(* Logix 5000 project; controller Uidaho_Factory vendor 1 type 14 code 165 rev 38.11; software revision 38.00 *)

TASK Heartbeat (periodic, rate 10000 ms, priority 10, watchdog 500 ms) : Heartbeat
TASK MainTask (continuous, watchdog 500 ms) : MainProgram

MODULES
   Local : vendor 1 type 14 code 165 (ICP 0, rev 38.11)
      Slot_3_Input : vendor 1 type 7 code 6 (ICP 3, rev 2.2, Input RPI 20 ms)
           Local:3:I.Data.3   // MPO - I8 = Reference switch vacuum (position oven)
           Local:3:I.Data.0   // MPO - I5 = Reference switch vacuum (position turn-table)
           Local:3:I.Data.5   // VGR - I1 = Reference switch vertical axis
           Local:3:I.Data.1   // MPO - I6 = Reference switch oven feeder inside
           Local:3:I.Data.2   // MPO - I7 = Reference switch oven feeder outside
           Local:3:I.Data.10   // SLD - I3 = Light barrier behind color sensor
           Local:3:I.Data.4   // MPO - I9 = Light barrier oven
           Local:3:I.Data.12   // SLD - I6 = Light barrier red
           Local:3:I.Data.13   // SLD - I7 = Light barrier blue
           Local:3:I.Data.8   // SLD - I1 = Pulse counter
           Local:3:I.Data.11   // SLD - I5 = Light barrier white
           Local:3:I.Data.9   // SLD - I2 = Light barrier inlet
           Local:3:I.Data.14   // SSC - I1 = Reference switch vertical axis
           Local:3:I.Data.6   // VGR - I2 = Reference switch horizontal axis
           Local:3:I.Data.7   // VGR - I3 = Reference switch rotate
           Local:3:I.Data.15   // SSC - I2 = Reference switch horizontal axis
      Slot_4_Input : vendor 1 type 7 code 6 (ICP 4, rev 2.2, Input RPI 20 ms)
           Local:4:I.Data.2   // SSC - B1 = Encoder vertical axis impulse 1
           Local:4:I.Data.1   // SSC - I4 = Light barrier behind color sensor
           Local:4:I.Data.4   // SSC - B3 = Encoder horizontal axis impulse 1
           Local:4:I.Data.5   // SSC - B4 = Encoder horizontal axis impulse 2
           Local:4:I.Data.3   // SSC - B2 = Encoder vertical axis impulse 2
           Local:4:I.Data.0   // SSC - I3 = Light barrier inlet
      Slot_2_Input : vendor 1 type 7 code 6 (ICP 2, rev 2.2, Input RPI 20 ms)
           Local:2:I.Data.15   // MPO - I4 = Reference switch turn-table (position saw)
           Local:2:I.Data.12   // MPO - I1 = Reference switch turn-table (position vacuum)
           Local:2:I.Data.3   // HBW - I4 = Reference switch vertical axis
           Local:2:I.Data.13   // MPO - I2 = Reference switch turn-table (position belt)
           Local:2:I.Data.14   // MPO - I3 = Light barrier end of conveyor belt
           Local:2:I.Data.10   // HBW - I5 = Reference switch cantilever front
           Local:2:I.Data.8   // HBW - B1 = Encoder horizontal axis impulse 1
           Local:2:I.Data.4   // HBW - A1 = Trail sensor (signal 1, lower)
           Local:2:I.Data.5   // HBW - A2 = Trail sensor (signal 2, upper)
           Local:2:I.Data.9   // HBW - B2 = Encoder horizontal axis impulse 2
           Local:2:I.Data.6   // HBW - B3 = Encoder vertical axis impulse 1
           Local:2:I.Data.7   // HBW - B4 = Encoder vertical axis impulse 2
           Local:2:I.Data.0   // HBW - I1 = Reference switch horizontal axis
           Local:2:I.Data.11   // HBW - I6 = Reference switch cantilever back
           Local:2:I.Data.2   // HBW - I3 = Light barrier outside
           Local:2:I.Data.1   // HBW - I2 = Light barrier inside
      Slot_1_Input : vendor 1 type 7 code 386 (ICP 1, rev 1.11, Output RPI 20 ms)
           Local:1:I.Pt[2].Data   // VGR - B3 = Encoder horizontal axis impulse 1
           Local:1:I.Pt[4].Data   // VGR - B5 = Encoder rotate impulse 1
           Local:1:I.Pt[5].Data   // VGR - B6 = Encoder rotate impulse 2
           Local:1:I.Pt[0].Data   // VGR - B1 = Encoder vertical axis impulse 1
           Local:1:I.Pt[3].Data   // VGR - B4 = Encoder horizontal axis impulse 2
           Local:1:I.Pt[1].Data   // VGR - B2 = Encoder vertical axis impulse 2
      Slot_6_Output : 1756-OB32 (ICP 6, rev 2.4, Output RPI 20 ms)
           Local:6:O.Data.17   // SSC - Q3 = Motor M2 horizontal axis backward
           Local:6:O.Data.20   // MPO - Q5 = Motor M4 oven feeder retract
           Local:6:O.Data.28   // VGR - Q3 = Motor M2 horizontal axis retract
           Local:6:O.Data.22   // MPO - Q2 = Motor M1 turn-table counterclockwise
           Local:6:O.Data.25   // MPO - Q10 = Compressor
           Local:6:O.Data.18   // SSC - Q4 = Motor M2 horizontal axis forward
           Local:6:O.Data.29   // VGR - Q4 = Motor M2 horizontal axis extend
           Local:6:O.Data.1   // HBW - Q6 = Motor M3 vertical axis upward
           Local:6:O.Data.10   // VGR - Q1 = Motor M1 vertical axis up
           Local:6:O.Data.11   // VGR - Q2 = Motor M1 vertical axis down
           Local:6:O.Data.9   // MPO - Q14 = Valve feeder
           Local:6:O.Data.16   // SSC - Q2 = Motor M1 vertical axis down
           Local:6:O.Data.2   // HBW - Q7 = Motor M4 cantilever forward
           Local:6:O.Data.30   // VGR - Q5 = Motor M3 rotate clockwise
           Local:6:O.Data.0   // HBW - Q5 = Motor M3 vertical axis downward
           Local:6:O.Data.4   // SSC = PWM Motor M1 vertical axis
           Local:6:O.Data.31   // VGR - Q6 = Motor M3 rotate counterclockwise
           Local:6:O.Data.3   // HBW - Q8 = Motor M4 cantilever backward
           Local:6:O.Data.14   // SLD - Q1 = Motor M1conveyor belt
           Local:6:O.Data.7   // MPO - Q8 = Motor M5 vacuum towards turn-table
           Local:6:O.Data.23   // MPO - Q3 = Motor M2 conveyor belt forward
           Local:6:O.Data.5   // SSC = PWM Motor M2 horizontal axis
           Local:6:O.Data.21   // MPO - Q1 = Motor M1 turn-table clockwise
           Local:6:O.Data.26   // MPO - Q11 = Valve vacuum
           Local:6:O.Data.19   // SSC - Q5 = LED Green
           Local:6:O.Data.27   // MPO - Q12 = Valve lowering
           Local:6:O.Data.13   // VGR - Q8 = Valve vacuum
           Local:6:O.Data.12   // VGR - Q7 = Compressor
           Local:6:O.Data.15   // SLD - Q2 = Compressor
           Local:6:O.Data.24   // MPO - Q9 = Light oven
           Local:6:O.Data.6   // QW_MPO_PWM_TurnTable_M1
           Local:6:O.Data.8   // MPO - Q13 = Valve oven door
      Slot_7_Output : 1756-OB32 (ICP 7, rev 3.2, Output RPI 20 ms)
           Local:7:O.Data.19   // VGR = PWM Motor M2 horizontal axis
           Local:7:O.Data.0   // SLD - Q3 = Valve first ejector (white)
           Local:7:O.Data.18   // VGR = PWM Motor M1 vertical axis
           Local:7:O.Data.3   // SSC - Q1 = Motor M1 vertical axis up
           Local:7:O.Data.1   // SLD - Q4 = Valve second ejector (red)
           Local:7:O.Data.15   // HBW = PWM Motor M2 horizontal axis
           Local:7:O.Data.12   // HBW - Q3 = Motor M2 horizontal towards rack
           Local:7:O.Data.13   // HBW - Q4 = Motor M2 horizontal towards conveyor belt
           Local:7:O.Data.8   // MPO - Q6 = Motor M4 oven feeder extend
           Local:7:O.Data.10   // HBW - Q1 = Motor M1 conveyor belt forward
           Local:7:O.Data.11   // HBW - Q2 = Motor M1 conveyor belt backward
           Local:7:O.Data.17   // HBW = PWM Motor M4 cantilever
           Local:7:O.Data.2   // SLD - Q5 = Valve third ejector (blue)
           Local:7:O.Data.21   // MPO = PWM Motor M5 vacuum
           Local:7:O.Data.9   // MPO - Q7 = Motor M5 vacuum towards oven
           Local:7:O.Data.20   // VGR = PWM Motor M3 rotate axis
           Local:7:O.Data.14   // HBW = PWM Motor M1 conveyor belt
           Local:7:O.Data.16   // HBW = PWM Motor M3 vertical axis
           Local:7:O.Data.6   // SSC - Q8 = LED Red Online
           Local:7:O.Data.7   // MPO - Q4 = Motor M3 saw
           Local:7:O.Data.4   // SSC - Q6 = LED Yellow
           Local:7:O.Data.5   // Turn on Motor Rotation Clockwise
      Slot_5_Input : 1756-IF8 (ICP 5, rev 1.5, Input RPI 100 ms)
           Local:5:I.Ch1Data   // SLD - A1 = Color sensor
           Local:5:I.Ch0Data   // SSC - A4 = Color sensor
END_MODULES

ADD_ON_INSTRUCTION PWM_Out   (* revision 1.0, ExecutePrescan *)
VAR_OUTPUT
   PWM_Pin : BOOL; {required}
END_VAR
VAR_INPUT
   Duty_Cycle : DINT; {required}
   Frequency_Hz : DINT; {required}
END_VAR
VAR
   PWM_Timer_On : TIMER; {access None}
   PWM_Timer_Off : TIMER; {access None}
   Duty_Cycle_Scaler : REAL; {access None}
   Frequency_Ms : REAL := 60.0; {access None}
   Fault_Bit : BOOL; {access None}
END_VAR

ROUTINE Logic   (* ladder *)
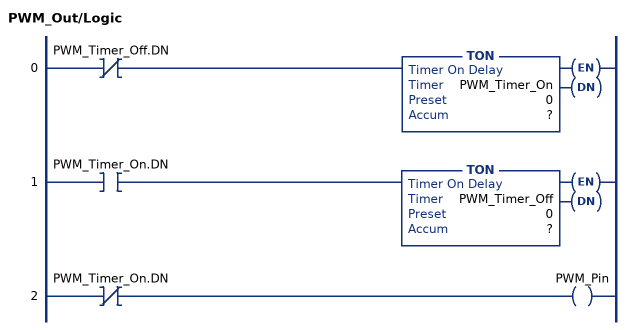
   0: XIO(PWM_Timer_Off.DN)TON(PWM_Timer_On,?,?);
   1: XIC(PWM_Timer_On.DN)TON(PWM_Timer_Off,?,?);
   2: XIO(PWM_Timer_On.DN)OTE(PWM_Pin);
END_ROUTINE

ROUTINE Prescan   (* ladder *)
// Perform Calculations for PWM Timing
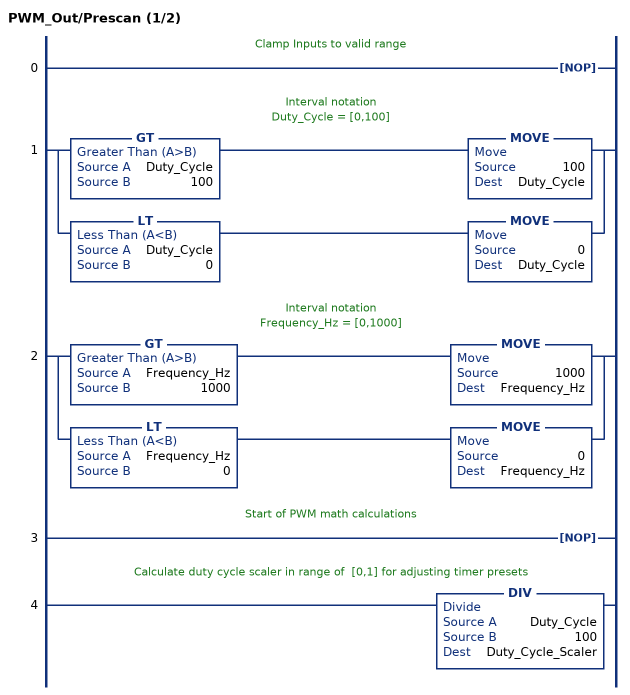
   // Clamp Inputs to valid range
   0: NOP();
   // Interval notation
   // Duty_Cycle = [0,100]
   1: [GT(Duty_Cycle,100) MOVE(100,Duty_Cycle) ,LT(Duty_Cycle,0) MOVE(0,Duty_Cycle) ];
   // Interval notation
   // Frequency_Hz = [0,1000]
   2: [GT(Frequency_Hz,1000) MOVE(1000,Frequency_Hz) ,LT(Frequency_Hz,0) MOVE(0,Frequency_Hz) ];
   // Start of PWM math calculations
   3: NOP();
   // Calculate duty cycle scaler in range of  [0,1] for adjusting timer presets
   4: DIV(Duty_Cycle,100,Duty_Cycle_Scaler);
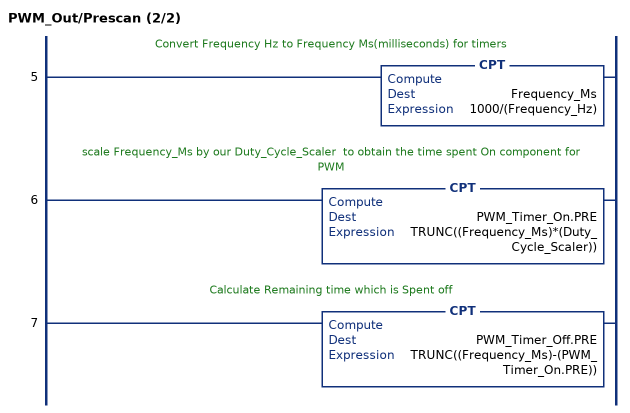
   // Convert Frequency Hz to Frequency Ms(milliseconds) for timers
   5: CPT(Frequency_Ms,1000/(Frequency_Hz));
   // scale Frequency_Ms by our Duty_Cycle_Scaler  to obtain the time spent On component for PWM
   6: CPT(PWM_Timer_On.PRE,TRUNC((Frequency_Ms)*(Duty_Cycle_Scaler)));
   // Calculate Remaining time which is Spent off
   7: CPT(PWM_Timer_Off.PRE,TRUNC((Frequency_Ms)-(PWM_Timer_On.PRE)));
END_ROUTINE
END_ADD_ON_INSTRUCTION

VAR_GLOBAL   (* controller tags *)
   Encoder_Counters_1X : COUNTER[10] := ([1].ACC := 690, [1].DN := 1, [2].DN := 1, [3].ACC := 5, [3].DN := 1, [4].PRE := 100, [4].ACC := 1345, [4].DN := 1);
        [4]   // VGR M3 Rotate 1X
        [0]   // HBW M2 Horizontal 1X
        [3]   // VGR M2 Horizontal 1X
        [1]   // HBW M3 Vertical 1X
        [2]   // VGR M1 Vertical 1X
   Encoder_Counters_2X : COUNTER[10] := ([0].ACC := -1927, [1].ACC := 697, [1].DN := 1, [2].ACC := 1, [2].DN := 1, [3].ACC := 5, [3].DN := 1, [4].ACC := 1345, [4].DN := 1);
        [4]   // VGR M3 Rotate 2X
        [0]   // HBW M2 Horizontal 2X
        [1]   // HBW M3 Vertical 2X
        [3]   // VGR M2 Horizontal 2X
        [2]   // VGR M1 Vertical 2X
   Encoder_Counters_4X : COUNTER[10] := ([1].ACC := 16114, [1].DN := 1, [2].ACC := -5907, [3].ACC := -1509, [4].PRE := 100, [4].ACC := 45779, [4].DN := 1);
        [4]   // VGR M3 Rotate 4X
        [0]   // HBW M2 Horizontal 4X
        [1]   // HBW M3 Vertical 4X
        [3]   // VGR M2 Horizontal 4X
        [2]   // VGR M1 Vertical 4X
   Encoder_Output_Bits_HBW : DINT;
   Encoder_Output_Bits_VGR : DINT[2];
   Encoder_Storage_Bits_HBW : DINT;
   Encoder_Storage_Bits_VGR : DINT[2];
   HBW_PWM_Outputs : PWM_Out[20] := ([0].PWM_Pin := 1, [0].Duty_Cycle := 100, [0].Frequency_Hz := 500, [1].PWM_Pin := 1, [1].Duty_Cycle := 100, [1].Frequency_Hz := 500, [2].PWM_Pin := 1, [2].Duty_Cycle := 100, [2].Frequency_Hz := 500, [3].PWM_Pin := 1, [3].Duty_Cycle := 100, [3].Frequency_Hz := 500);
   HeartbeatError : BOOL;
   I_O_Counter : COUNTER[20] := ([0].PRE := 2140000000, [1].PRE := 2140000000, [2].PRE := 2140000000, [3].PRE := 2140000000, [4].PRE := 2140000000, [4].ACC := 2, [5].PRE := 2140000000, [6].PRE := 2140000000, [6].ACC := 42, [9].PRE := 2140000000, [9].CU := 1);
   PWM_Outputs : PWM_Out[20] := ([0].Duty_Cycle := 100, [0].Frequency_Hz := 500, [1].Duty_Cycle := 100, [1].Frequency_Hz := 500, [2].Duty_Cycle := 100, [2].Frequency_Hz := 500, [3].Duty_Cycle := 100, [3].Frequency_Hz := 500, [4].PWM_Pin := 1, [4].Duty_Cycle := 100, [4].Frequency_Hz := 500, [5].PWM_Pin := 1, [5].Duty_Cycle := 100, [5].Frequency_Hz := 500, [6].PWM_Pin := 1, [6].Duty_Cycle := 100, [6].Frequency_Hz := 500, [7].PWM_Pin := 1, [7].Duty_Cycle := 100, [7].Frequency_Hz := 500, [8].PWM_Pin := 1, [8].Duty_Cycle := 100, [8].Frequency_Hz := 500, [9].Duty_Cycle := 100, [9].Frequency_Hz := 500, [10].Duty_Cycle := 100, [10].Frequency_Hz := 500);
   Scaled_Analog_Color_Sensor_SLD : DINT := 38256;   // SLD - A1 = Color sensor
   Slot_1_Faulted : DINT;
   Slot_2_Faulted : DINT;
   Slot_3_Faulted : DINT;
   Slot_4_Faulted : DINT;
   Slot_5_Faulted : DINT;
   Slot_6_Faulted : DINT;
   Slot_7_Faulted : DINT;
   Slot_9_Faulted : DINT;
   VGR_PWM_Outputs : PWM_Out[20] := ([8].PWM_Pin := 1, [8].Duty_Cycle := 100, [8].Frequency_Hz := 500, [9].PWM_Pin := 1, [9].Duty_Cycle := 100, [9].Frequency_Hz := 500, [10].PWM_Pin := 1, [10].Duty_Cycle := 100, [10].Frequency_Hz := 500);
END_VAR

PROGRAM Heartbeat   (* main routine Heartbeat *)
VAR
   HeartbeatCurrent : DINT;
   HeartbeatOld : DINT;
END_VAR

ROUTINE Heartbeat   (* ladder *)
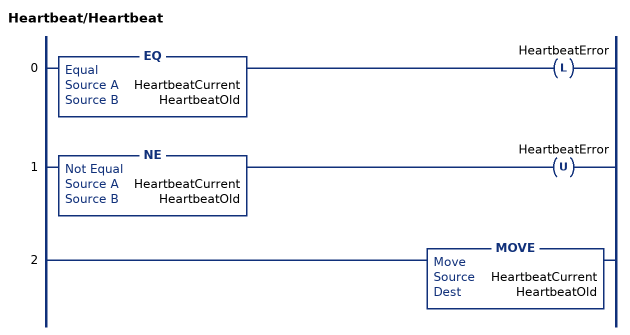
   0: EQ(HeartbeatCurrent,HeartbeatOld)OTL(HeartbeatError);
   1: NE(HeartbeatCurrent,HeartbeatOld)OTU(HeartbeatError);
   2: MOVE(HeartbeatCurrent,HeartbeatOld);
END_ROUTINE
END_PROGRAM

PROGRAM MainProgram   (* main routine MainRoutine *)
VAR
   ESTOP : BOOL;
   Fault_Detected : BOOL;   // On if an issue of any sort happens. Estop, connection failure, safety device activation, etc...
   GripperTimers : TIMER[10] := ([0].PRE := 1000, [1].PRE := 1000, [2].PRE := 1000, [3].PRE := 1000, [4].PRE := 1000, [5].PRE := 1000);
   Homing : BOOL;
   MPO_Auto : BOOL;
   MPO_Compressor_Button : BOOL;
   MPO_Conveyor_Button : BOOL;
   MPO_Done : BOOL;
   MPO_Feeder_Extend_Button : BOOL;
   MPO_Feeder_Retract_Button : BOOL;
   MPO_Gripper_Direction_Manual : BOOL;   // 0 - positive 1 - negative
   MPO_Gripper_Lower_Button : BOOL;
   MPO_Gripper_On : BOOL;   // 0 - Off 1 - On
   MPO_Gripper_Piston : BOOL;   // 0 - retracted 1- extended
   MPO_Gripper_Start : BOOL;
   MPO_Gripper_Toward_Oven_Button : BOOL;
   MPO_Gripper_Toward_Table_Button : BOOL;
   MPO_Gripper_Valve_Button : BOOL;
   MPO_Has_Puck : BOOL;
   MPO_Homing : BOOL;
   MPO_Jog_Gripper : BOOL;   // 0 - no movement 1 - movement
   MPO_Jog_Oven_Door : BOOL;   // 0 - no movement 1- movement
   MPO_Jog_Oven_Table : BOOL;   // 0 - no movement 1 - movement
   MPO_Jog_Saw : BOOL;   // 0 - off 1 - on
   MPO_Jog_Turntable : BOOL;   // 0 - no movement 1 - movement
   MPO_Oven_Door_Button : BOOL;
   MPO_Oven_Door_Direction : BOOL;   // 0 - negative 1 - positive
   MPO_Oven_Light_Button : BOOL;
   MPO_Oven_On : BOOL;   // 0 - off 1 - on
   MPO_Oven_Start : BOOL;
   MPO_Oven_Table_Direction : BOOL;   // 0 - negative 1 - positive
   MPO_Saw_Button : BOOL;
   MPO_Turntable_CCW_Button : BOOL;
   MPO_Turntable_CW_Button : BOOL;
   MPO_Turntable_Direction : BOOL;   // 0 - negative 1 - positive
   MPO_Turntable_Piston : BOOL;   // 0 - retracted 1 - extended
   MPO_Turntable_Pusher_Button : BOOL;
   MPO_Turntable_Start : BOOL;
   Operation_Mode : DINT := 1;   // 0 - Off 1 - Manual 2 - Automatic
   OvenTimers : TIMER[10] := ([0].PRE := 1000, [1].PRE := 1000, [2].PRE := 3000, [3].PRE := 1000, [4].PRE := 1000);
   SCL_01 : SCALE := (In := 5.837123, InRawMax := 10.0, InEUMax := 65535.0, Out := 38253.586);   // Scaler for SLD - A1 = Color sensor
   SLD_Blue_Min : DINT := 34000; {constant}
   SLD_Blue_Time : DINT := 2460; {constant}
   SLD_Jog_Belt : BOOL;   // 0 - dont run 1 - run
   SLD_Jog_Blue_Piston : BOOL;   // 0 - retracted 1 - extended
   SLD_Jog_Red_Piston : BOOL;   // 0 - retracted 1 - extended
   SLD_Jog_White_Piston : BOOL;   // 0 - retracted 1 - extended
   SLD_Min_Value : DINT := 36000;
   SLD_Move_Puck_To_Sensor_Time : DINT := 1800; {constant}
   SLD_Move_Time : DINT := 1420;
   SLD_Normal : DINT := 38000; {constant}
   SLD_Red_Min : DINT := 18000; {constant}
   SLD_Red_Time : DINT := 1420; {constant}
   SLD_start : DINT;
   SLD_Step : DINT;
   SLD_White_Min : DINT; {constant}
   SLD_White_Time : DINT := 438; {constant}
   Start : DINT;
   Step : DINT[20];
   StepTimers : TIMER[20] := ([0].PRE := 2000, [1].PRE := 1420, [3].PRE := 1000);
   TurntableTimers : TIMER[10] := ([0].PRE := 3000, [1].PRE := 1000);
END_VAR

ROUTINE Analog_Scaling   (* function block diagram *)
   SHEET 1
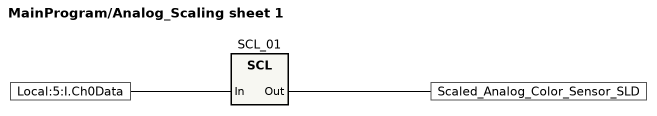
   SCL_01 : SCL(In := Local:5:I.Ch0Data);
   Scaled_Analog_Color_Sensor_SLD := SCL_01.Out;
END_ROUTINE

ROUTINE AutomaticRoutine   (* ladder *)
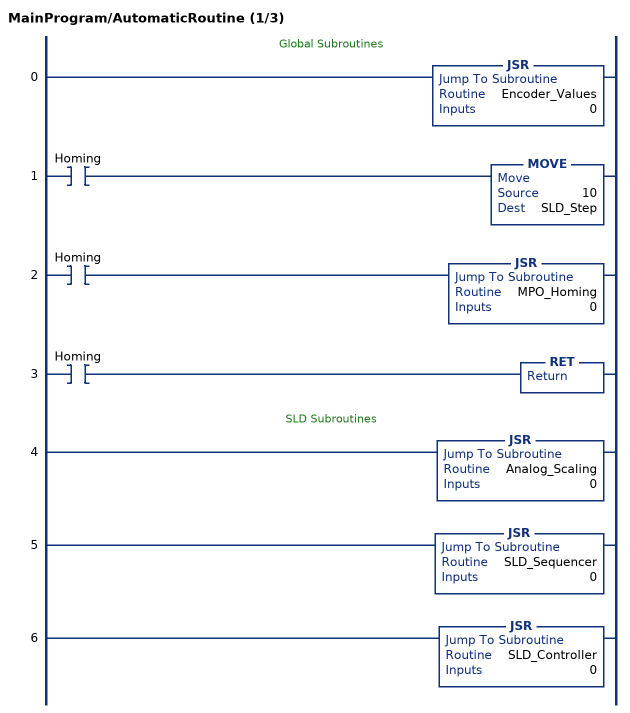
   // Global Subroutines
   0: JSR(Encoder_Values,0);
   1: XIC(Homing)MOVE(10,SLD_Step);
   2: XIC(Homing)JSR(MPO_Homing,0);
   3: XIC(Homing)RET();
   // SLD Subroutines
   4: JSR(Analog_Scaling,0);
   5: JSR(SLD_Sequencer,0);
   6: JSR(SLD_Controller,0);
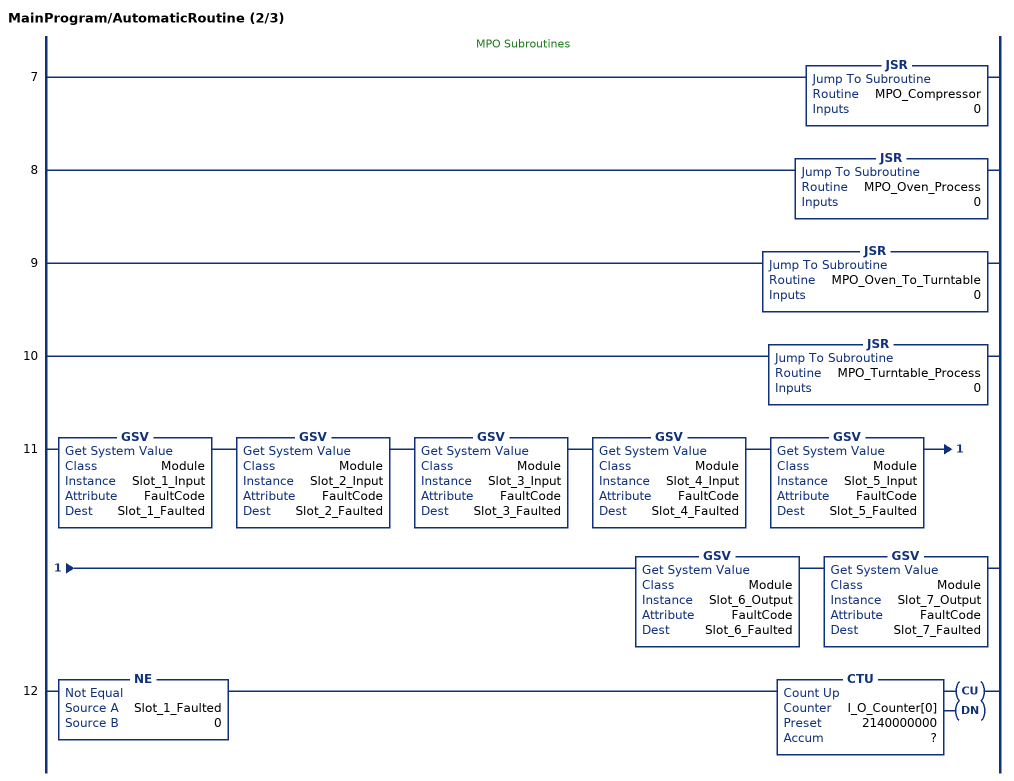
   // MPO Subroutines
   7: JSR(MPO_Compressor,0);
   8: JSR(MPO_Oven_Process,0);
   9: JSR(MPO_Oven_To_Turntable,0);
   10: JSR(MPO_Turntable_Process,0);
   11: GSV(Module,Slot_1_Input,FaultCode,Slot_1_Faulted)GSV(Module,Slot_2_Input,FaultCode,Slot_2_Faulted)GSV(Module,Slot_3_Input,FaultCode,Slot_3_Faulted)GSV(Module,Slot_4_Input,FaultCode,Slot_4_Faulted)GSV(Module,Slot_5_Input,FaultCode,Slot_5_Faulted)GSV(Module,Slot_6_Output,FaultCode,Slot_6_Faulted)GSV(Module,Slot_7_Output,FaultCode,Slot_7_Faulted);
   12: NE(Slot_1_Faulted,0)CTU(I_O_Counter[0],?,?);
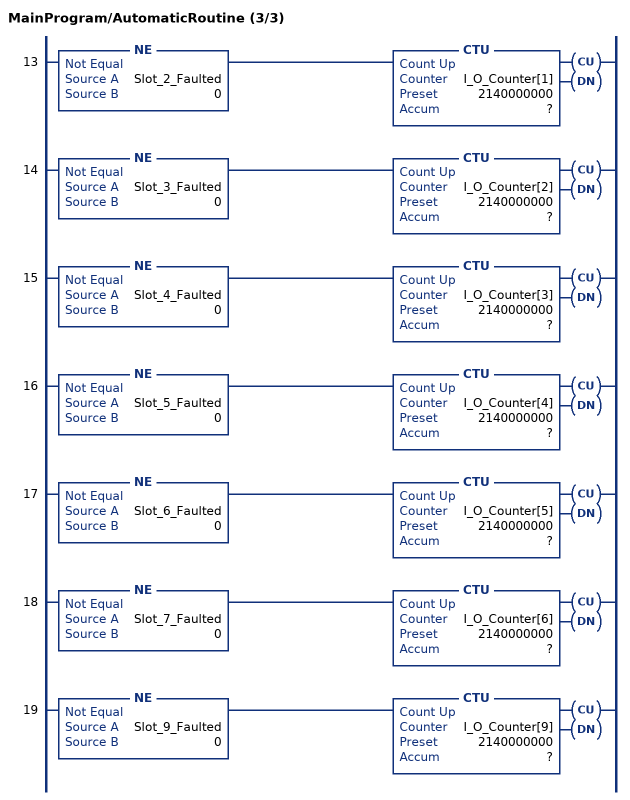
   13: NE(Slot_2_Faulted,0)CTU(I_O_Counter[1],?,?);
   14: NE(Slot_3_Faulted,0)CTU(I_O_Counter[2],?,?);
   15: NE(Slot_4_Faulted,0)CTU(I_O_Counter[3],?,?);
   16: NE(Slot_5_Faulted,0)CTU(I_O_Counter[4],?,?);
   17: NE(Slot_6_Faulted,0)CTU(I_O_Counter[5],?,?);
   18: NE(Slot_7_Faulted,0)CTU(I_O_Counter[6],?,?);
   19: NE(Slot_9_Faulted,0)CTU(I_O_Counter[9],?,?);
END_ROUTINE

ROUTINE Encoder_Values   (* ladder *)
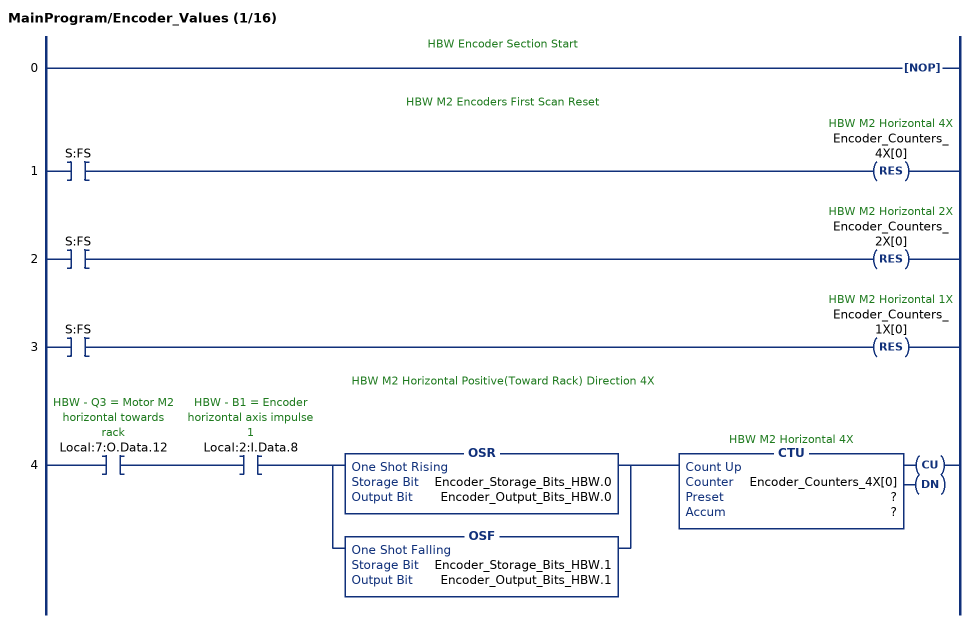
   // HBW Encoder Section Start
   0: NOP();
   // HBW M2 Encoders First Scan Reset
   1: XIC(S:FS)RES(Encoder_Counters_4X[0]);
   2: XIC(S:FS)RES(Encoder_Counters_2X[0]);
   3: XIC(S:FS)RES(Encoder_Counters_1X[0]);
   // HBW M2 Horizontal Positive(Toward Rack) Direction 4X
   4: XIC(Local:7:O.Data.12)XIC(Local:2:I.Data.8)[OSR(Encoder_Storage_Bits_HBW.0,Encoder_Output_Bits_HBW.0) ,OSF(Encoder_Storage_Bits_HBW.1,Encoder_Output_Bits_HBW.1) ]CTU(Encoder_Counters_4X[0],?,?);
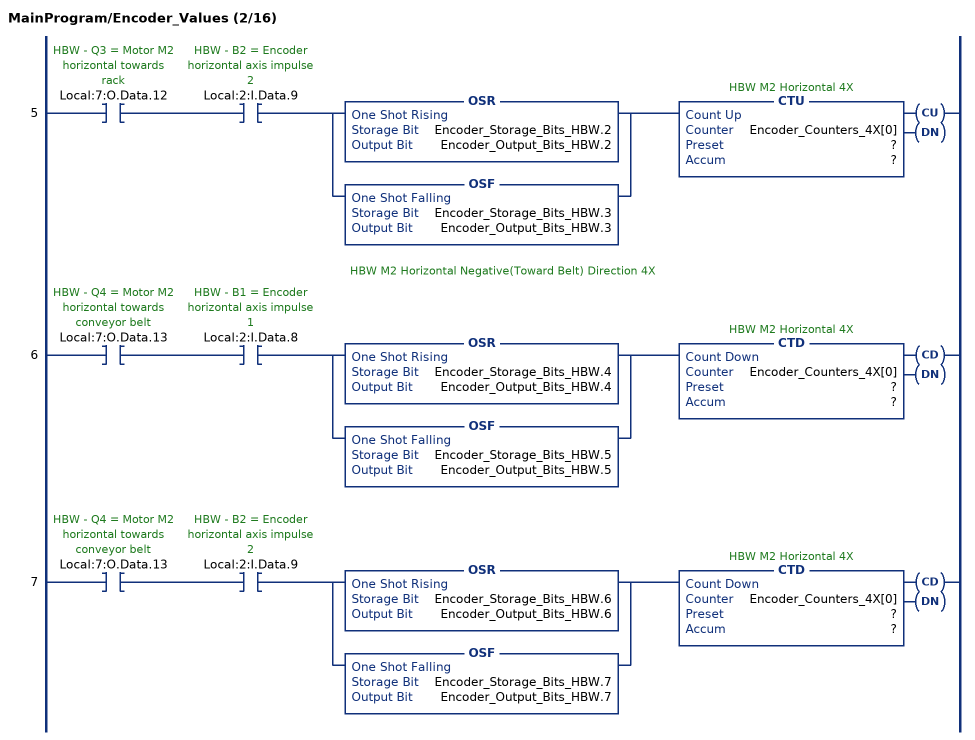
   5: XIC(Local:7:O.Data.12)XIC(Local:2:I.Data.9)[OSR(Encoder_Storage_Bits_HBW.2,Encoder_Output_Bits_HBW.2) ,OSF(Encoder_Storage_Bits_HBW.3,Encoder_Output_Bits_HBW.3) ]CTU(Encoder_Counters_4X[0],?,?);
   // HBW M2 Horizontal Negative(Toward Belt) Direction 4X
   6: XIC(Local:7:O.Data.13)XIC(Local:2:I.Data.8)[OSR(Encoder_Storage_Bits_HBW.4,Encoder_Output_Bits_HBW.4) ,OSF(Encoder_Storage_Bits_HBW.5,Encoder_Output_Bits_HBW.5) ]CTD(Encoder_Counters_4X[0],?,?);
   7: XIC(Local:7:O.Data.13)XIC(Local:2:I.Data.9)[OSR(Encoder_Storage_Bits_HBW.6,Encoder_Output_Bits_HBW.6) ,OSF(Encoder_Storage_Bits_HBW.7,Encoder_Output_Bits_HBW.7) ]CTD(Encoder_Counters_4X[0],?,?);
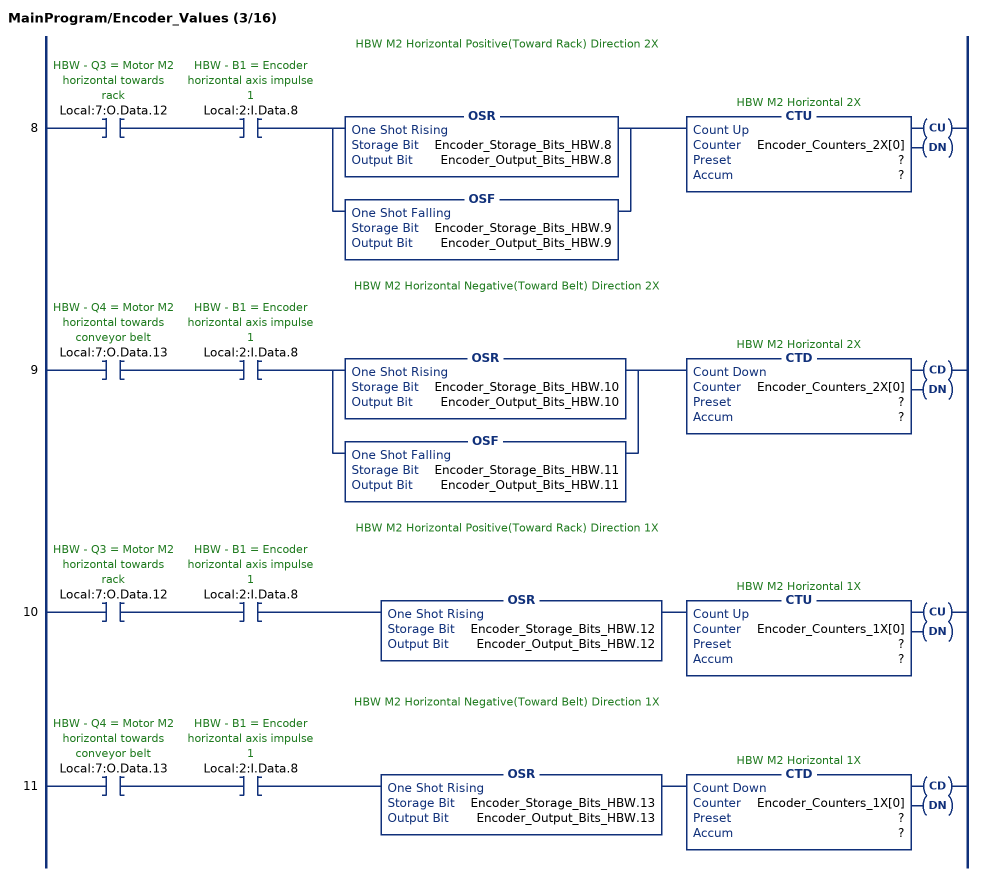
   // HBW M2 Horizontal Positive(Toward Rack) Direction 2X
   8: XIC(Local:7:O.Data.12)XIC(Local:2:I.Data.8)[OSR(Encoder_Storage_Bits_HBW.8,Encoder_Output_Bits_HBW.8) ,OSF(Encoder_Storage_Bits_HBW.9,Encoder_Output_Bits_HBW.9) ]CTU(Encoder_Counters_2X[0],?,?);
   // HBW M2 Horizontal Negative(Toward Belt) Direction 2X
   9: XIC(Local:7:O.Data.13)XIC(Local:2:I.Data.8)[OSR(Encoder_Storage_Bits_HBW.10,Encoder_Output_Bits_HBW.10) ,OSF(Encoder_Storage_Bits_HBW.11,Encoder_Output_Bits_HBW.11) ]CTD(Encoder_Counters_2X[0],?,?);
   // HBW M2 Horizontal Positive(Toward Rack) Direction 1X
   10: XIC(Local:7:O.Data.12)XIC(Local:2:I.Data.8)OSR(Encoder_Storage_Bits_HBW.12,Encoder_Output_Bits_HBW.12)CTU(Encoder_Counters_1X[0],?,?);
   // HBW M2 Horizontal Negative(Toward Belt) Direction 1X
   11: XIC(Local:7:O.Data.13)XIC(Local:2:I.Data.8)OSR(Encoder_Storage_Bits_HBW.13,Encoder_Output_Bits_HBW.13)CTD(Encoder_Counters_1X[0],?,?);
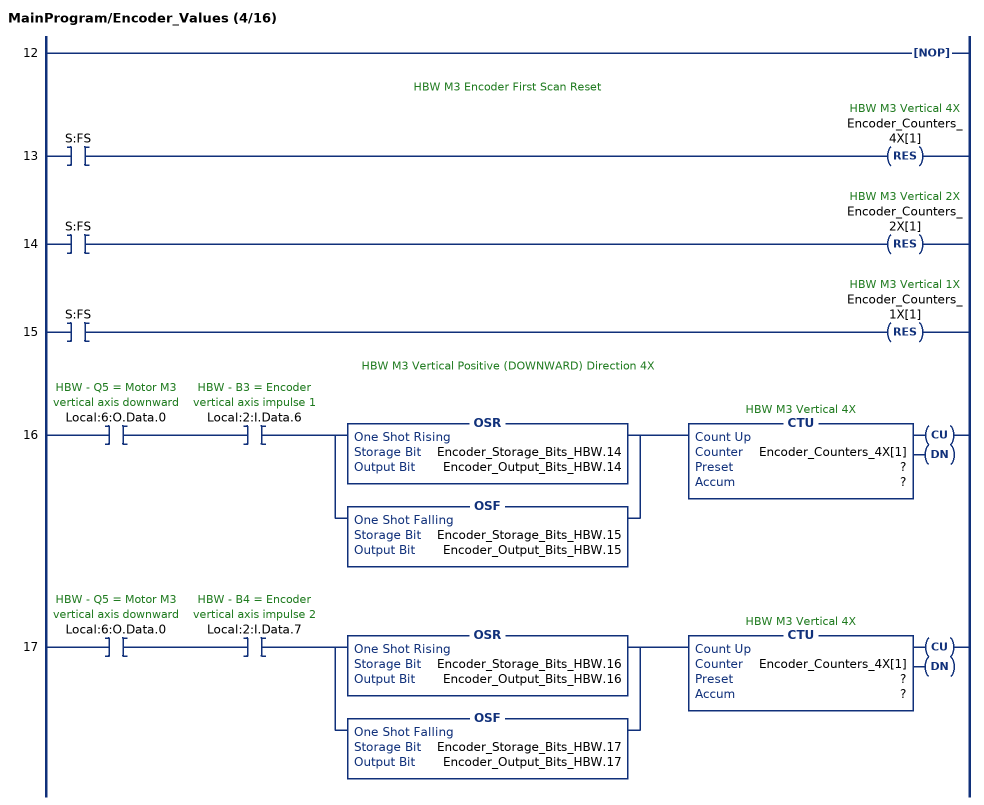
   12: NOP();
   // HBW M3 Encoder First Scan Reset
   13: XIC(S:FS)RES(Encoder_Counters_4X[1]);
   14: XIC(S:FS)RES(Encoder_Counters_2X[1]);
   15: XIC(S:FS)RES(Encoder_Counters_1X[1]);
   // HBW M3 Vertical Positive (DOWNWARD) Direction 4X
   16: XIC(Local:6:O.Data.0)XIC(Local:2:I.Data.6)[OSR(Encoder_Storage_Bits_HBW.14,Encoder_Output_Bits_HBW.14) ,OSF(Encoder_Storage_Bits_HBW.15,Encoder_Output_Bits_HBW.15) ]CTU(Encoder_Counters_4X[1],?,?);
   17: XIC(Local:6:O.Data.0)XIC(Local:2:I.Data.7)[OSR(Encoder_Storage_Bits_HBW.16,Encoder_Output_Bits_HBW.16) ,OSF(Encoder_Storage_Bits_HBW.17,Encoder_Output_Bits_HBW.17) ]CTU(Encoder_Counters_4X[1],?,?);
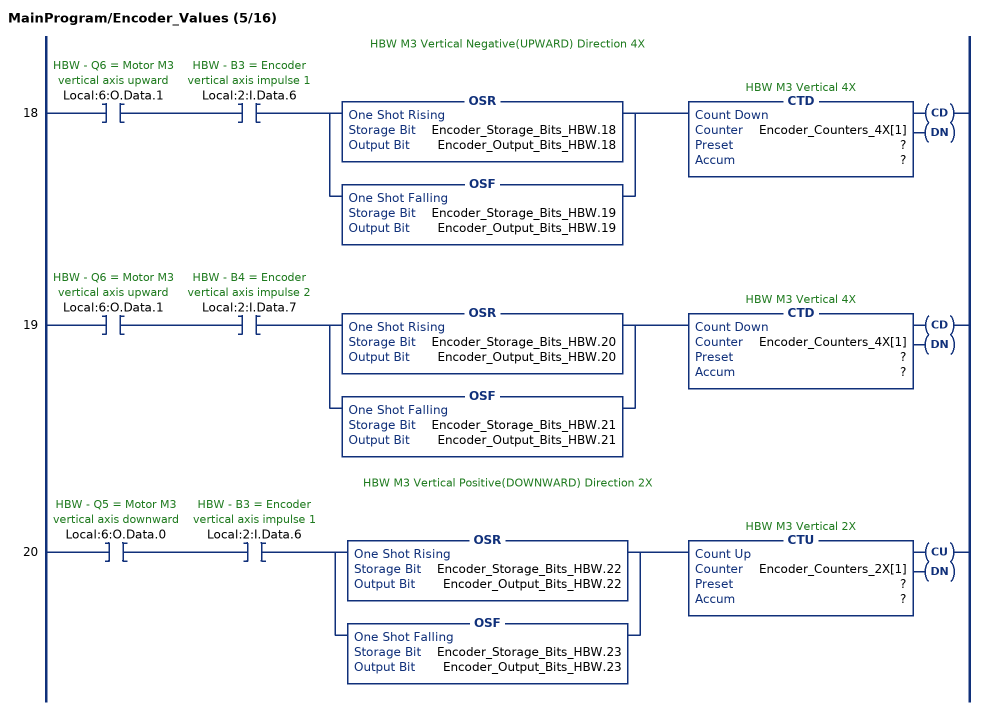
   // HBW M3 Vertical Negative(UPWARD) Direction 4X
   18: XIC(Local:6:O.Data.1)XIC(Local:2:I.Data.6)[OSR(Encoder_Storage_Bits_HBW.18,Encoder_Output_Bits_HBW.18) ,OSF(Encoder_Storage_Bits_HBW.19,Encoder_Output_Bits_HBW.19) ]CTD(Encoder_Counters_4X[1],?,?);
   19: XIC(Local:6:O.Data.1)XIC(Local:2:I.Data.7)[OSR(Encoder_Storage_Bits_HBW.20,Encoder_Output_Bits_HBW.20) ,OSF(Encoder_Storage_Bits_HBW.21,Encoder_Output_Bits_HBW.21) ]CTD(Encoder_Counters_4X[1],?,?);
   // HBW M3 Vertical Positive(DOWNWARD) Direction 2X
   20: XIC(Local:6:O.Data.0)XIC(Local:2:I.Data.6)[OSR(Encoder_Storage_Bits_HBW.22,Encoder_Output_Bits_HBW.22) ,OSF(Encoder_Storage_Bits_HBW.23,Encoder_Output_Bits_HBW.23) ]CTU(Encoder_Counters_2X[1],?,?);
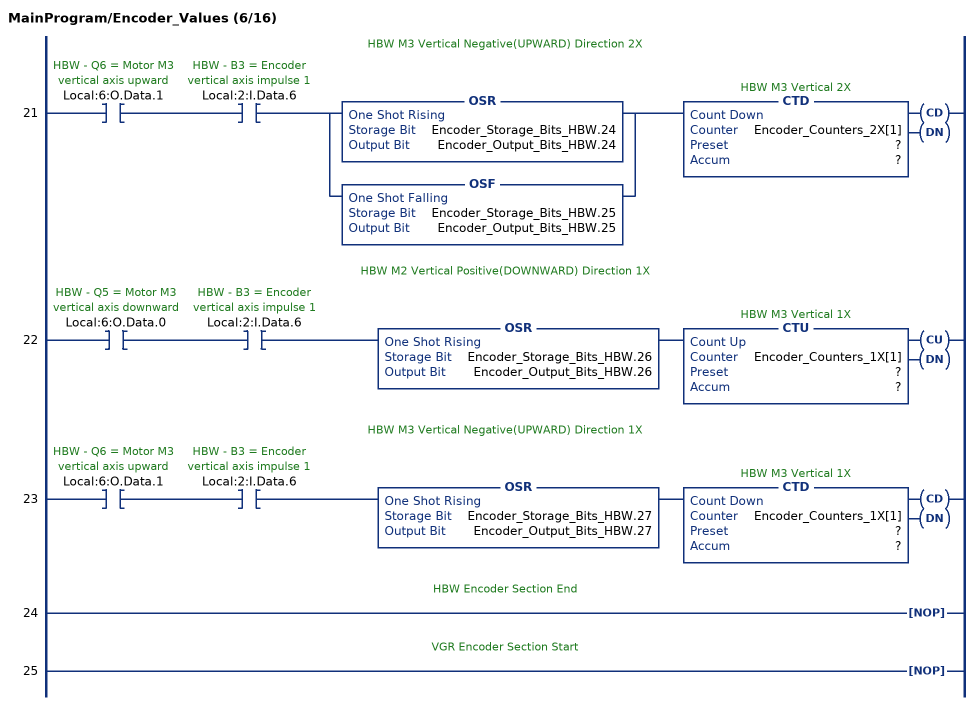
   // HBW M3 Vertical Negative(UPWARD) Direction 2X
   21: XIC(Local:6:O.Data.1)XIC(Local:2:I.Data.6)[OSR(Encoder_Storage_Bits_HBW.24,Encoder_Output_Bits_HBW.24) ,OSF(Encoder_Storage_Bits_HBW.25,Encoder_Output_Bits_HBW.25) ]CTD(Encoder_Counters_2X[1],?,?);
   // HBW M2 Vertical Positive(DOWNWARD) Direction 1X
   22: XIC(Local:6:O.Data.0)XIC(Local:2:I.Data.6)OSR(Encoder_Storage_Bits_HBW.26,Encoder_Output_Bits_HBW.26)CTU(Encoder_Counters_1X[1],?,?);
   // HBW M3 Vertical Negative(UPWARD) Direction 1X
   23: XIC(Local:6:O.Data.1)XIC(Local:2:I.Data.6)OSR(Encoder_Storage_Bits_HBW.27,Encoder_Output_Bits_HBW.27)CTD(Encoder_Counters_1X[1],?,?);
   // HBW Encoder Section End
   24: NOP();
   // VGR Encoder Section Start
   25: NOP();
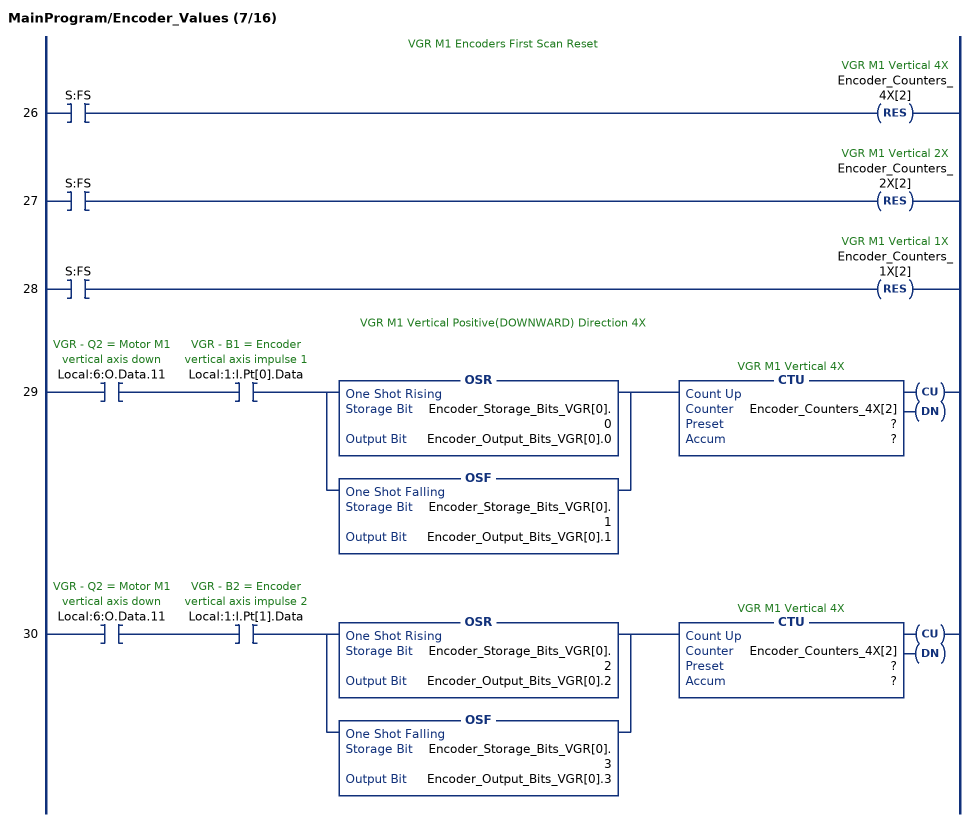
   // VGR M1 Encoders First Scan Reset
   26: XIC(S:FS)RES(Encoder_Counters_4X[2]);
   27: XIC(S:FS)RES(Encoder_Counters_2X[2]);
   28: XIC(S:FS)RES(Encoder_Counters_1X[2]);
   // VGR M1 Vertical Positive(DOWNWARD) Direction 4X
   29: XIC(Local:6:O.Data.11)XIC(Local:1:I.Pt[0].Data)[OSR(Encoder_Storage_Bits_VGR[0].0,Encoder_Output_Bits_VGR[0].0) ,OSF(Encoder_Storage_Bits_VGR[0].1,Encoder_Output_Bits_VGR[0].1) ]CTU(Encoder_Counters_4X[2],?,?);
   30: XIC(Local:6:O.Data.11)XIC(Local:1:I.Pt[1].Data)[OSR(Encoder_Storage_Bits_VGR[0].2,Encoder_Output_Bits_VGR[0].2) ,OSF(Encoder_Storage_Bits_VGR[0].3,Encoder_Output_Bits_VGR[0].3) ]CTU(Encoder_Counters_4X[2],?,?);
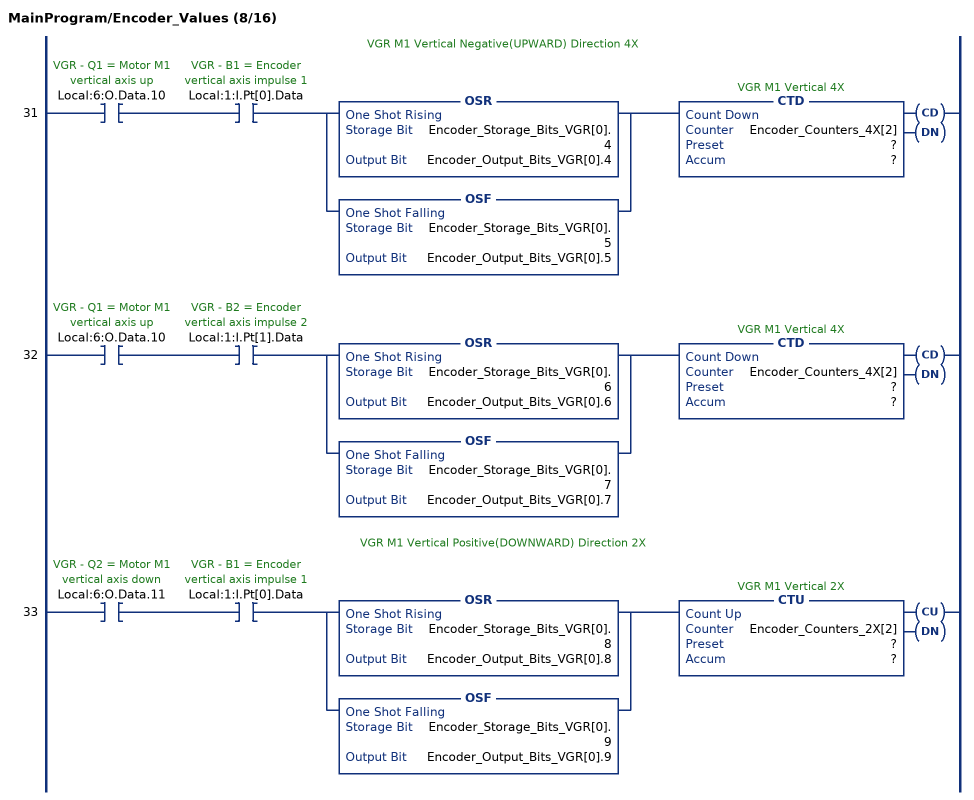
   // VGR M1 Vertical Negative(UPWARD) Direction 4X
   31: XIC(Local:6:O.Data.10)XIC(Local:1:I.Pt[0].Data)[OSR(Encoder_Storage_Bits_VGR[0].4,Encoder_Output_Bits_VGR[0].4) ,OSF(Encoder_Storage_Bits_VGR[0].5,Encoder_Output_Bits_VGR[0].5) ]CTD(Encoder_Counters_4X[2],?,?);
   32: XIC(Local:6:O.Data.10)XIC(Local:1:I.Pt[1].Data)[OSR(Encoder_Storage_Bits_VGR[0].6,Encoder_Output_Bits_VGR[0].6) ,OSF(Encoder_Storage_Bits_VGR[0].7,Encoder_Output_Bits_VGR[0].7) ]CTD(Encoder_Counters_4X[2],?,?);
   // VGR M1 Vertical Positive(DOWNWARD) Direction 2X
   33: XIC(Local:6:O.Data.11)XIC(Local:1:I.Pt[0].Data)[OSR(Encoder_Storage_Bits_VGR[0].8,Encoder_Output_Bits_VGR[0].8) ,OSF(Encoder_Storage_Bits_VGR[0].9,Encoder_Output_Bits_VGR[0].9) ]CTU(Encoder_Counters_2X[2],?,?);
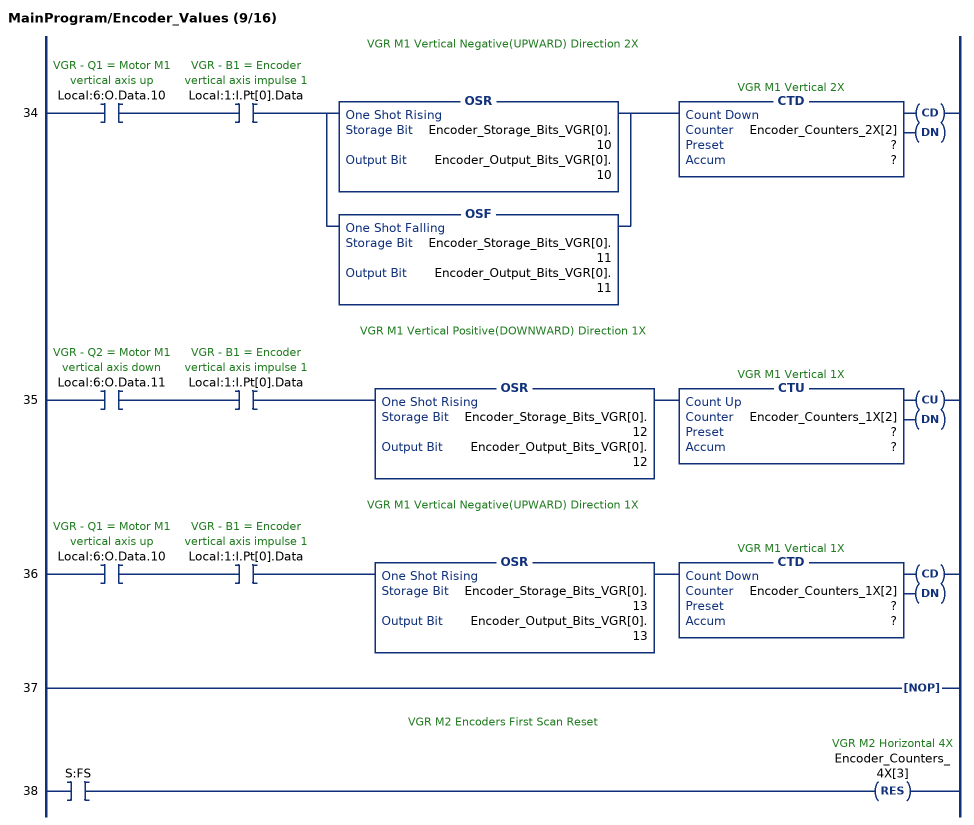
   // VGR M1 Vertical Negative(UPWARD) Direction 2X
   34: XIC(Local:6:O.Data.10)XIC(Local:1:I.Pt[0].Data)[OSR(Encoder_Storage_Bits_VGR[0].10,Encoder_Output_Bits_VGR[0].10) ,OSF(Encoder_Storage_Bits_VGR[0].11,Encoder_Output_Bits_VGR[0].11) ]CTD(Encoder_Counters_2X[2],?,?);
   // VGR M1 Vertical Positive(DOWNWARD) Direction 1X
   35: XIC(Local:6:O.Data.11)XIC(Local:1:I.Pt[0].Data)OSR(Encoder_Storage_Bits_VGR[0].12,Encoder_Output_Bits_VGR[0].12)CTU(Encoder_Counters_1X[2],?,?);
   // VGR M1 Vertical Negative(UPWARD) Direction 1X
   36: XIC(Local:6:O.Data.10)XIC(Local:1:I.Pt[0].Data)OSR(Encoder_Storage_Bits_VGR[0].13,Encoder_Output_Bits_VGR[0].13)CTD(Encoder_Counters_1X[2],?,?);
   37: NOP();
   // VGR M2 Encoders First Scan Reset
   38: XIC(S:FS)RES(Encoder_Counters_4X[3]);
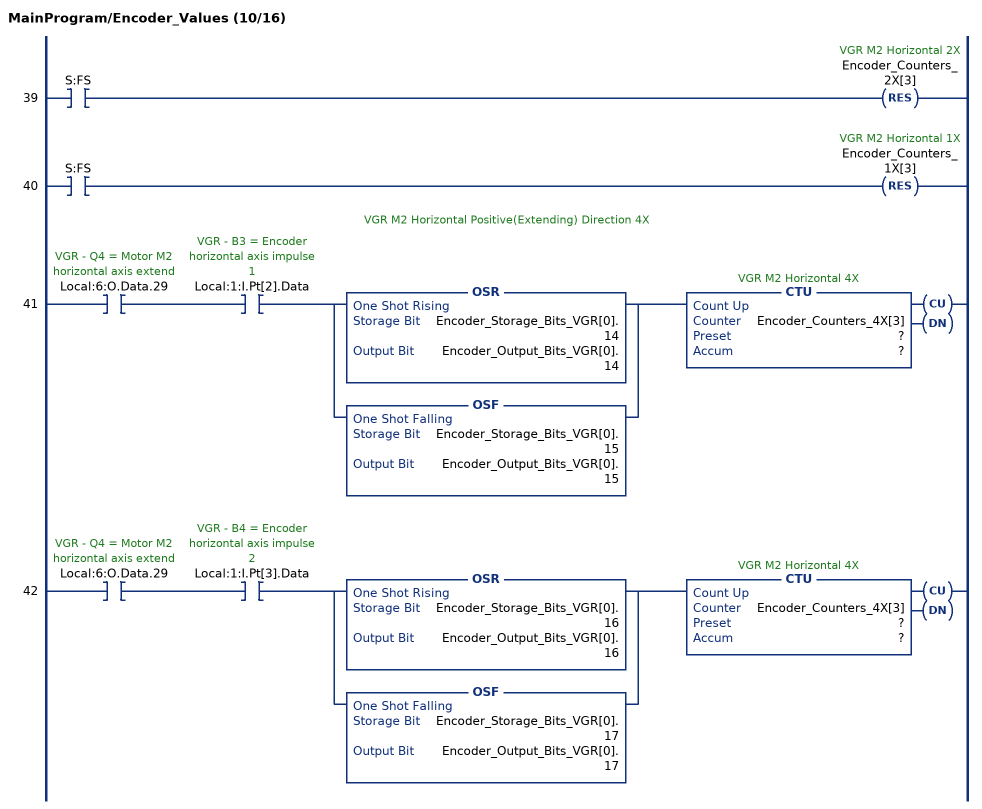
   39: XIC(S:FS)RES(Encoder_Counters_2X[3]);
   40: XIC(S:FS)RES(Encoder_Counters_1X[3]);
   // VGR M2 Horizontal Positive(Extending) Direction 4X
   41: XIC(Local:6:O.Data.29)XIC(Local:1:I.Pt[2].Data)[OSR(Encoder_Storage_Bits_VGR[0].14,Encoder_Output_Bits_VGR[0].14) ,OSF(Encoder_Storage_Bits_VGR[0].15,Encoder_Output_Bits_VGR[0].15) ]CTU(Encoder_Counters_4X[3],?,?);
   42: XIC(Local:6:O.Data.29)XIC(Local:1:I.Pt[3].Data)[OSR(Encoder_Storage_Bits_VGR[0].16,Encoder_Output_Bits_VGR[0].16) ,OSF(Encoder_Storage_Bits_VGR[0].17,Encoder_Output_Bits_VGR[0].17) ]CTU(Encoder_Counters_4X[3],?,?);
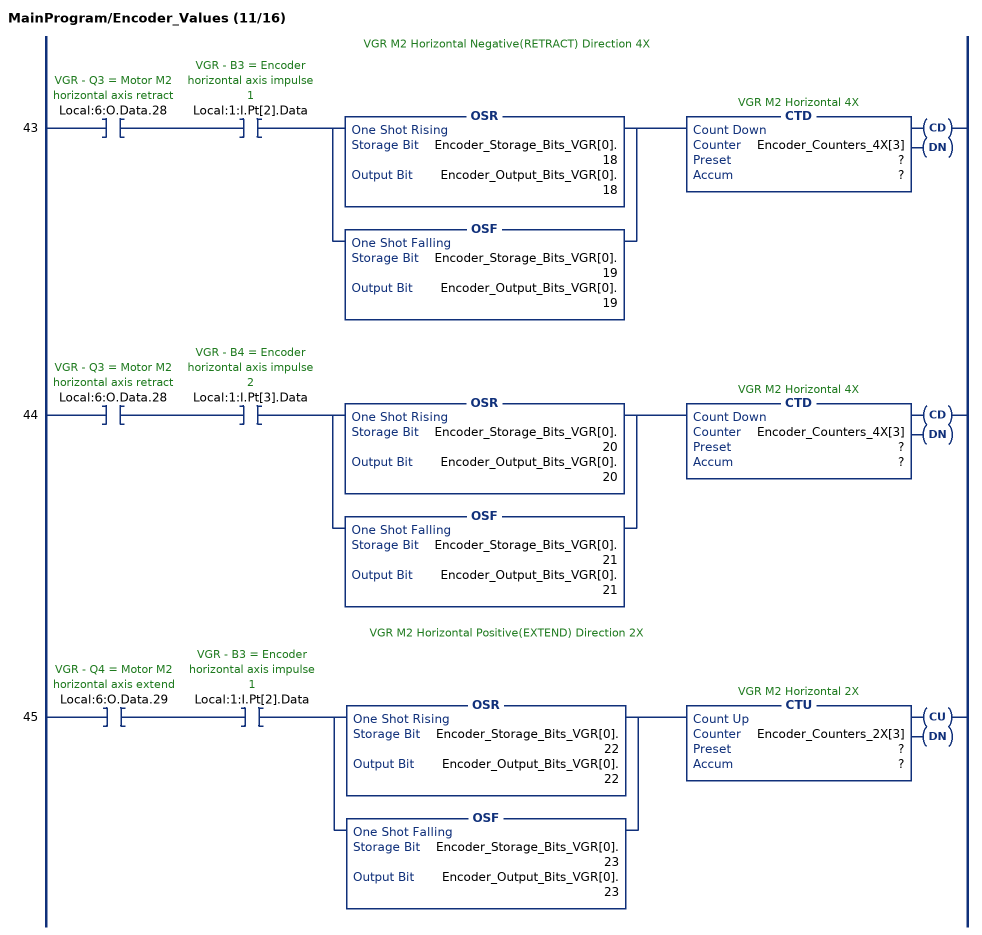
   // VGR M2 Horizontal Negative(RETRACT) Direction 4X
   43: XIC(Local:6:O.Data.28)XIC(Local:1:I.Pt[2].Data)[OSR(Encoder_Storage_Bits_VGR[0].18,Encoder_Output_Bits_VGR[0].18) ,OSF(Encoder_Storage_Bits_VGR[0].19,Encoder_Output_Bits_VGR[0].19) ]CTD(Encoder_Counters_4X[3],?,?);
   44: XIC(Local:6:O.Data.28)XIC(Local:1:I.Pt[3].Data)[OSR(Encoder_Storage_Bits_VGR[0].20,Encoder_Output_Bits_VGR[0].20) ,OSF(Encoder_Storage_Bits_VGR[0].21,Encoder_Output_Bits_VGR[0].21) ]CTD(Encoder_Counters_4X[3],?,?);
   // VGR M2 Horizontal Positive(EXTEND) Direction 2X
   45: XIC(Local:6:O.Data.29)XIC(Local:1:I.Pt[2].Data)[OSR(Encoder_Storage_Bits_VGR[0].22,Encoder_Output_Bits_VGR[0].22) ,OSF(Encoder_Storage_Bits_VGR[0].23,Encoder_Output_Bits_VGR[0].23) ]CTU(Encoder_Counters_2X[3],?,?);
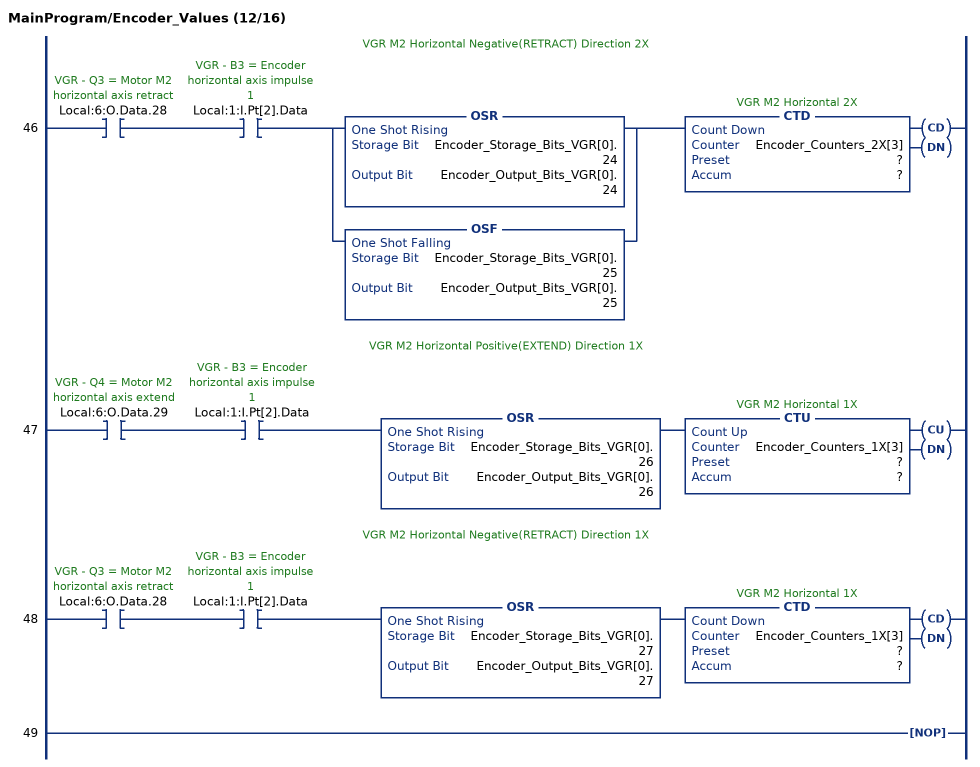
   // VGR M2 Horizontal Negative(RETRACT) Direction 2X
   46: XIC(Local:6:O.Data.28)XIC(Local:1:I.Pt[2].Data)[OSR(Encoder_Storage_Bits_VGR[0].24,Encoder_Output_Bits_VGR[0].24) ,OSF(Encoder_Storage_Bits_VGR[0].25,Encoder_Output_Bits_VGR[0].25) ]CTD(Encoder_Counters_2X[3],?,?);
   // VGR M2 Horizontal Positive(EXTEND) Direction 1X
   47: XIC(Local:6:O.Data.29)XIC(Local:1:I.Pt[2].Data)OSR(Encoder_Storage_Bits_VGR[0].26,Encoder_Output_Bits_VGR[0].26)CTU(Encoder_Counters_1X[3],?,?);
   // VGR M2 Horizontal Negative(RETRACT) Direction 1X
   48: XIC(Local:6:O.Data.28)XIC(Local:1:I.Pt[2].Data)OSR(Encoder_Storage_Bits_VGR[0].27,Encoder_Output_Bits_VGR[0].27)CTD(Encoder_Counters_1X[3],?,?);
   49: NOP();
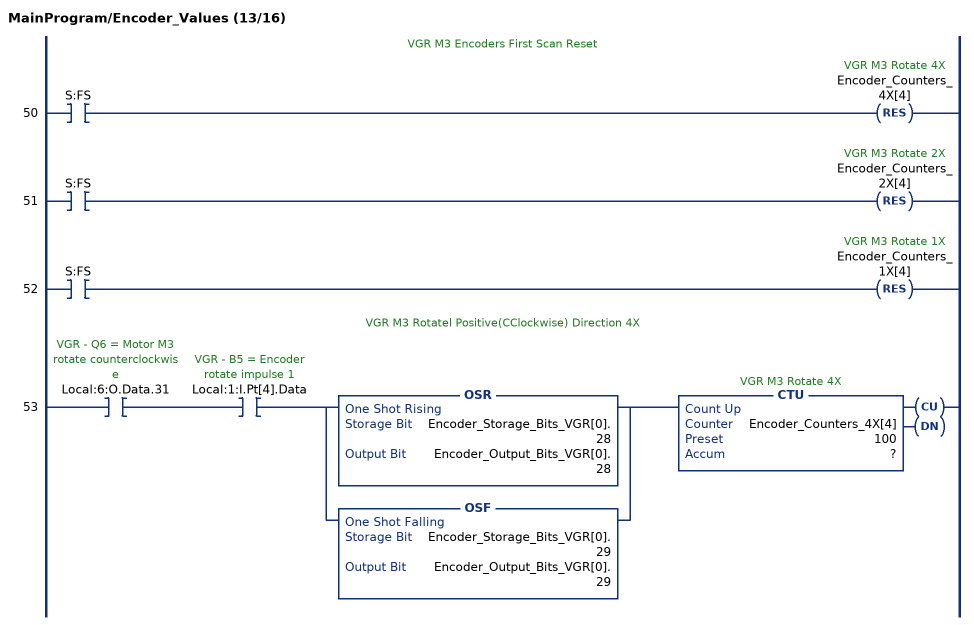
   // VGR M3 Encoders First Scan Reset
   50: XIC(S:FS)RES(Encoder_Counters_4X[4]);
   51: XIC(S:FS)RES(Encoder_Counters_2X[4]);
   52: XIC(S:FS)RES(Encoder_Counters_1X[4]);
   // VGR M3 Rotatel Positive(CClockwise) Direction 4X
   53: XIC(Local:6:O.Data.31)XIC(Local:1:I.Pt[4].Data)[OSR(Encoder_Storage_Bits_VGR[0].28,Encoder_Output_Bits_VGR[0].28) ,OSF(Encoder_Storage_Bits_VGR[0].29,Encoder_Output_Bits_VGR[0].29) ]CTU(Encoder_Counters_4X[4],?,?);
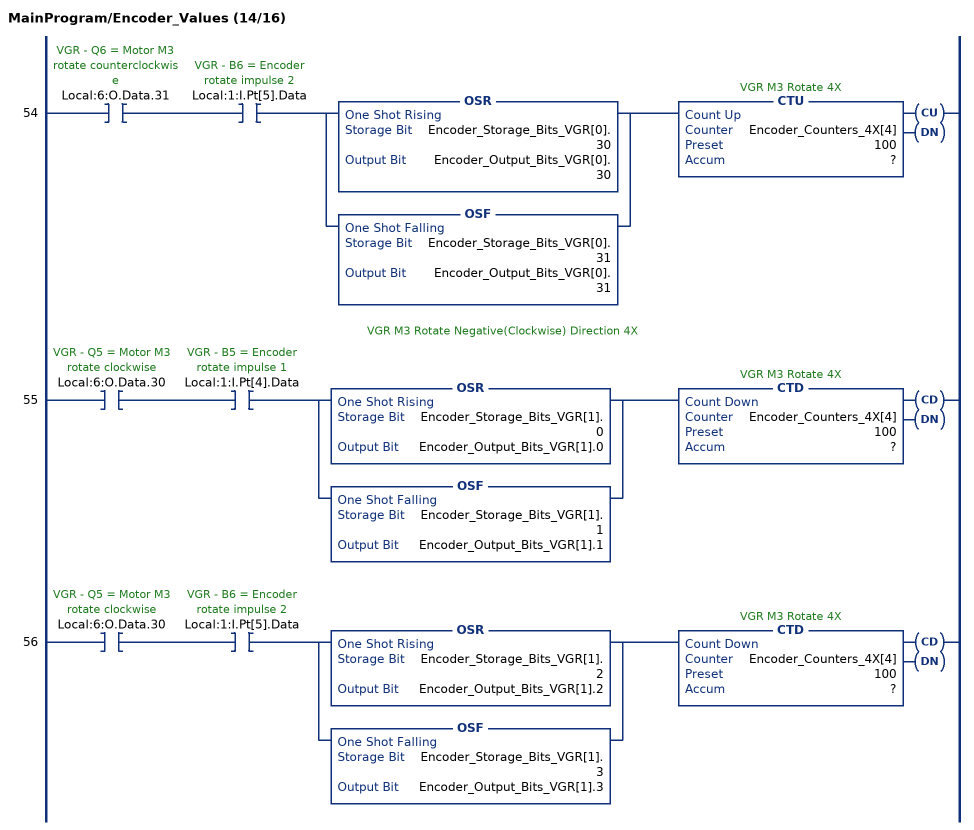
   54: XIC(Local:6:O.Data.31)XIC(Local:1:I.Pt[5].Data)[OSR(Encoder_Storage_Bits_VGR[0].30,Encoder_Output_Bits_VGR[0].30) ,OSF(Encoder_Storage_Bits_VGR[0].31,Encoder_Output_Bits_VGR[0].31) ]CTU(Encoder_Counters_4X[4],?,?);
   // VGR M3 Rotate Negative(Clockwise) Direction 4X
   55: XIC(Local:6:O.Data.30)XIC(Local:1:I.Pt[4].Data)[OSR(Encoder_Storage_Bits_VGR[1].0,Encoder_Output_Bits_VGR[1].0) ,OSF(Encoder_Storage_Bits_VGR[1].1,Encoder_Output_Bits_VGR[1].1) ]CTD(Encoder_Counters_4X[4],?,?);
   56: XIC(Local:6:O.Data.30)XIC(Local:1:I.Pt[5].Data)[OSR(Encoder_Storage_Bits_VGR[1].2,Encoder_Output_Bits_VGR[1].2) ,OSF(Encoder_Storage_Bits_VGR[1].3,Encoder_Output_Bits_VGR[1].3) ]CTD(Encoder_Counters_4X[4],?,?);
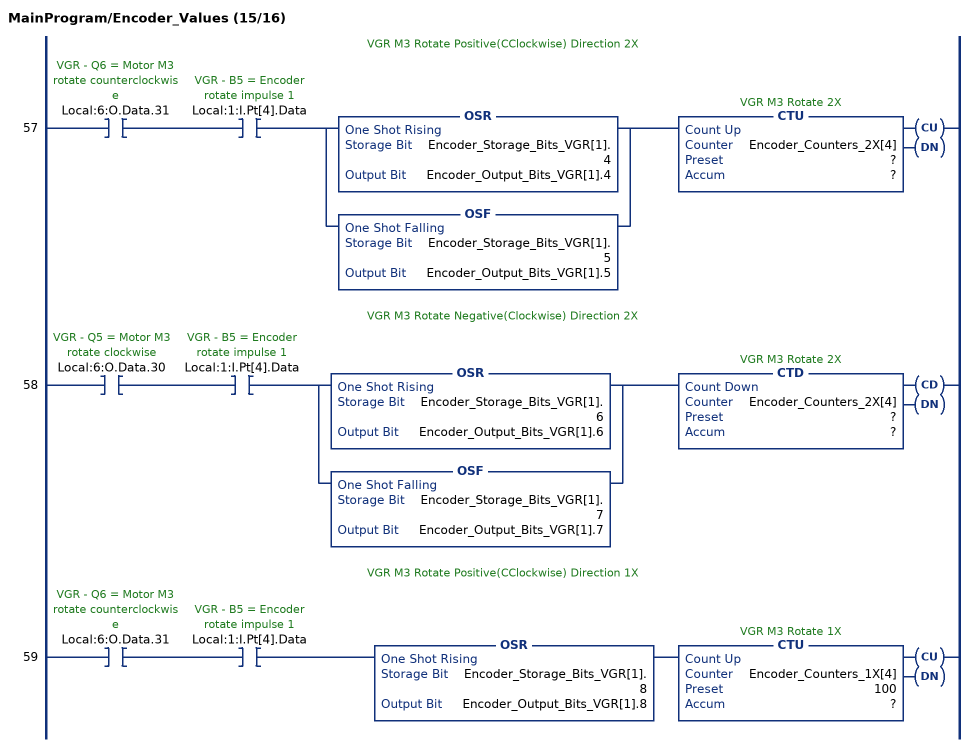
   // VGR M3 Rotate Positive(CClockwise) Direction 2X
   57: XIC(Local:6:O.Data.31)XIC(Local:1:I.Pt[4].Data)[OSR(Encoder_Storage_Bits_VGR[1].4,Encoder_Output_Bits_VGR[1].4) ,OSF(Encoder_Storage_Bits_VGR[1].5,Encoder_Output_Bits_VGR[1].5) ]CTU(Encoder_Counters_2X[4],?,?);
   // VGR M3 Rotate Negative(Clockwise) Direction 2X
   58: XIC(Local:6:O.Data.30)XIC(Local:1:I.Pt[4].Data)[OSR(Encoder_Storage_Bits_VGR[1].6,Encoder_Output_Bits_VGR[1].6) ,OSF(Encoder_Storage_Bits_VGR[1].7,Encoder_Output_Bits_VGR[1].7) ]CTD(Encoder_Counters_2X[4],?,?);
   // VGR M3 Rotate Positive(CClockwise) Direction 1X
   59: XIC(Local:6:O.Data.31)XIC(Local:1:I.Pt[4].Data)OSR(Encoder_Storage_Bits_VGR[1].8,Encoder_Output_Bits_VGR[1].8)CTU(Encoder_Counters_1X[4],?,?);
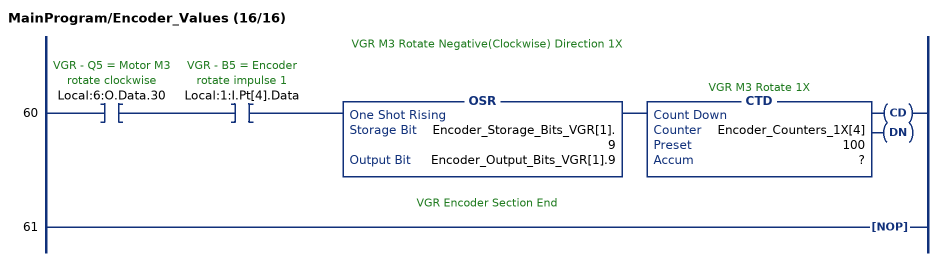
   // VGR M3 Rotate Negative(Clockwise) Direction 1X
   60: XIC(Local:6:O.Data.30)XIC(Local:1:I.Pt[4].Data)OSR(Encoder_Storage_Bits_VGR[1].9,Encoder_Output_Bits_VGR[1].9)CTD(Encoder_Counters_1X[4],?,?);
   // VGR Encoder Section End
   61: NOP();
END_ROUTINE
